FUNCTION_BLOCK SUBL_105_DRILLING-ROUND_HOLE (* 105-variable local group subscriber *)
  (* Standard: 61499-2 *)
  (* Version 1.0, 21-03-12, GASR, Universidade do Estado de Santa Catarina *)
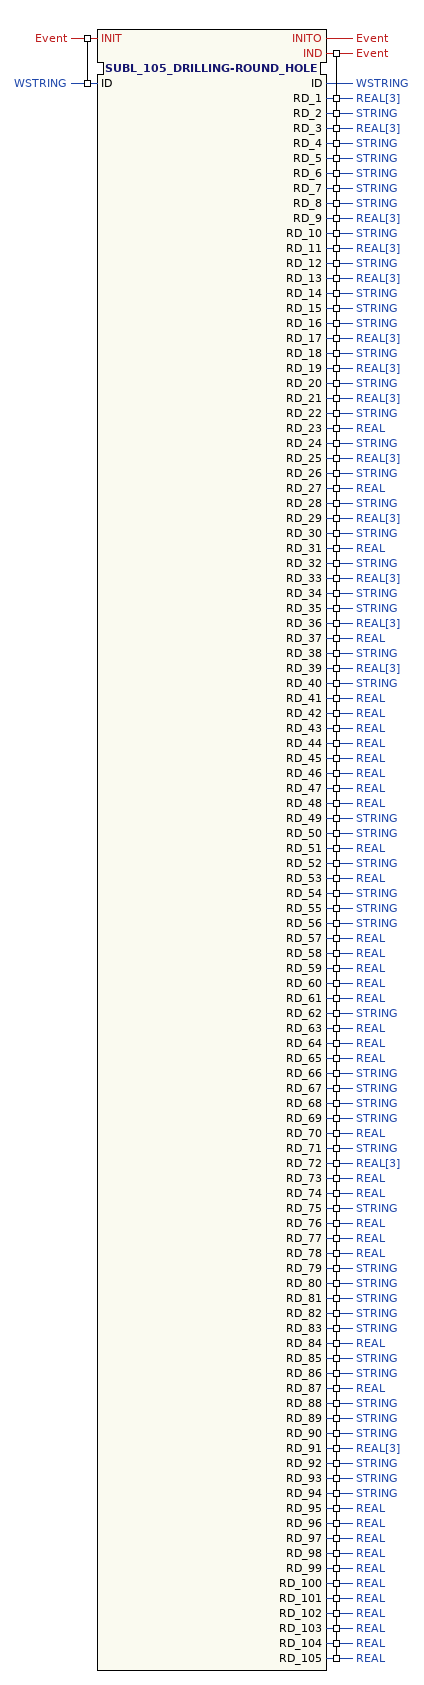
  EVENT_INPUT
    INIT WITH ID; (* Service Initialization *)
  END_EVENT
  EVENT_OUTPUT
    INITO; (* Initialization Confirm *)
    IND WITH RD_1, RD_2, RD_3, RD_4, RD_5, RD_6, RD_7, RD_8, RD_9, RD_10, RD_11, RD_12, RD_13, RD_14, RD_15, RD_16, RD_17, RD_18, RD_19, RD_20, RD_21, RD_22, RD_23, RD_24, RD_25, RD_26, RD_27, RD_28, RD_29, RD_30, RD_31, RD_32, RD_33, RD_34, RD_35, RD_36, RD_37, RD_38, RD_39, RD_40, RD_41, RD_42, RD_43, RD_44, RD_45, RD_46, RD_47, RD_48, RD_49, RD_50, RD_51, RD_52, RD_53, RD_54, RD_55, RD_56, RD_57, RD_58, RD_59, RD_60, RD_61, RD_62, RD_63, RD_64, RD_65, RD_66, RD_67, RD_68, RD_69, RD_70, RD_71, RD_72, RD_73, RD_74, RD_75, RD_76, RD_77, RD_78, RD_79, RD_80, RD_81, RD_82, RD_83, RD_84, RD_85, RD_86, RD_87, RD_88, RD_89, RD_90, RD_91, RD_92, RD_93, RD_94, RD_95, RD_96, RD_97, RD_98, RD_99, RD_100, RD_101, RD_102, RD_103, RD_104, RD_105; (* Service Indication *)
  END_EVENT
  VAR_INPUT
    ID : WSTRING; (* Default id is the FB instance name *)
  END_VAR
  VAR_OUTPUT
    ID : WSTRING; (* Default id is the FB instance name *)
    RD_1 : ARRAY [0..2] OF REAL; (* pos *)
    RD_2 : STRING; (* current_tool *)
    RD_3 : ARRAY [0..2] OF REAL; (* setup.Its_secplane.position.location.coordinates *)
    RD_4 : STRING; (* round_hole.its_id *)
    RD_5 : STRING; (* its_workpiece.its_id *)
    RD_6 : STRING; (* its_operations.its_id LIST - the list is concatenated in one string *)
    RD_7 : STRING; (* feature_placement.name *)
    RD_8 : STRING; (* feature_placement.location.name *)
    RD_9 : ARRAY [0..2] OF REAL; (* feature_placement.location.coordinates *)
    RD_10 : STRING; (* feature_placement.axis.its_id *)
    RD_11 : ARRAY [0..2] OF REAL; (* feature_placement.axis.direction_ratios *)
    RD_12 : STRING; (* feature_placement.ref_direction.its_id *)
    RD_13 : ARRAY [0..2] OF REAL; (* feature_placement.ref_direction_ratios *)
    RD_14 : STRING; (* depth.name *)
    RD_15 : STRING; (* depth.postion.name *)
    RD_16 : STRING; (* depth.position.location.name *)
    RD_17 : ARRAY [0..2] OF REAL; (* depth.position.location.coordinates *)
    RD_18 : STRING; (* depth.position.axis.its_id *)
    RD_19 : ARRAY [0..2] OF REAL; (* depth.position.axis.direction_ratios *)
    RD_20 : STRING; (* depth.position.ref_direction.its_id *)
    RD_21 : ARRAY [0..2] OF REAL; (* depth.position.ref_direction_ratios *)
    RD_22 : STRING; (* diameter *)
    RD_23 : REAL; (* diameter.theoretical_size *)
    RD_24 : STRING; (* diameter.implicit_tolerance *)
    RD_25 : ARRAY [0..2] OF REAL; (* diameter.{vector}, vector = {upper_limit, lower_limit, significant_digits} or {deviation,grade,its_fitting_type} *)
    RD_26 : STRING; (* change_in_diameter, "diameter_taper" or "angle_taper" *)
    RD_27 : REAL; (* change_in_diameter.theoretical_size *)
    RD_28 : STRING; (* change_in_diameter.implicit_tolerance *)
    RD_29 : ARRAY [0..2] OF REAL; (* change_in_diameter.{vector}, vector = {upper_limit, lower_limit, significant_digits} or {deviation,grade,its_fitting_type} *)
    RD_30 : STRING; (* bottom_condition, "through_bottom_condition" or ... *)
    RD_31 : REAL; (* bottom_condition.theoretical_size *)
    RD_32 : STRING; (* bottom_condition.implicit_tolerance *)
    RD_33 : ARRAY [0..2] OF REAL; (* bottom_condition.{vector}, vector = {upper_limit, lower_limit, significant_digits} or {deviation,grade,its_fitting_type} *)
    RD_34 : STRING; (* drilling.its_id *)
    RD_35 : STRING; (* its_toolpath.its_list *)
    RD_36 : ARRAY [0..2] OF REAL; (* its_tool_direction *)
    RD_37 : REAL; (* retract_plane *)
    RD_38 : STRING; (* start_point.name *)
    RD_39 : ARRAY [0..2] OF REAL; (* start_point.coordinates *)
    RD_40 : STRING; (* its_tool.its_id *)
    RD_41 : REAL; (* its_tool.its_tool_body.dimension.diameter *)
    RD_42 : REAL; (* its_tool.its_tool_body.dimension.tool_tip_half_angle *)
    RD_43 : REAL; (* its_tool.its_tool_body.dimension.tool_circumference_angle *)
    RD_44 : REAL; (* its_tool.its_tool_body.dimension.cutting_edge_lenght *)
    RD_45 : REAL; (* its_tool.its_tool_body.dimension.edge_radius *)
    RD_46 : REAL; (* its_tool.its_tool_body.dimension.edge_center_vertical *)
    RD_47 : REAL; (* its_tool.its_tool_body.dimension.edge_center_horizontal *)
    RD_48 : REAL; (* its_tool.its_tool_body.number_of_teeth *)
    RD_49 : STRING; (* its_tool.its_tool_body.hand_of_cut *)
    RD_50 : STRING; (* its_tool.its_tool_body.coolant_through *)
    RD_51 : REAL; (* its_tool.its_tool_body.pilot_length *)
    RD_52 : STRING; (* its_tool.its_tool_body.{other_tool_body_parameter} *)
    RD_53 : REAL; (* its_tool.its_cutting_edge.tool_offset_length *)
    RD_54 : STRING; (* its_tool.its_cutting_edge.its_material.standard_identifier *)
    RD_55 : STRING; (* its_tool.its_cutting_edge.its_material.material_identifier *)
    RD_56 : STRING; (* its_tool.its_cutting_edge.its_material.material_property.{list_of_parameters} *)
    RD_57 : REAL; (* its_tool.its_cutting_edge.its_technological_data.cutting_angle *)
    RD_58 : REAL; (* its_tool.its_cutting_edge.its_technological_data.free_angle *)
    RD_59 : REAL; (* its_tool.its_cutting_edge.its_technological_data.aux_angle *)
    RD_60 : REAL; (* its_tool.its_cutting_edge.expected_tool_life *)
    RD_61 : REAL; (* its_tool.its_cutting_edge.its_technology.feedrate *)
    RD_62 : STRING; (* its_tool.its_cutting_edge.its_technology.feedrate_reference *)
    RD_63 : REAL; (* its_tool.its_cutting_edge.its_technology.cutspeed *)
    RD_64 : REAL; (* its_tool.its_cutting_edge.its_technology.spindle *)
    RD_65 : REAL; (* its_tool.its_cutting_edge.its_technology.feedrate_per_tooth *)
    RD_66 : STRING; (* its_tool.its_cutting_edge.its_technology.sincronize_spindle_with_feed *)
    RD_67 : STRING; (* its_tool.its_cutting_edge.its_technology.inhibit_feedrate_override *)
    RD_68 : STRING; (* its_tool.its_cutting_edge.its_technology.inhibit_spindle_override *)
    RD_69 : STRING; (* its_tool.its_cutting_edge.its_technology.its_adaptive_control *)
    RD_70 : REAL; (* its_tool.overall_assembly_length *)
    RD_71 : STRING; (* its_tool.direction_for_spindle_orientation.its_id *)
    RD_72 : ARRAY [0..2] OF REAL; (* its_tool.direction_for_spindle_orientation.direction_ratios *)
    RD_73 : REAL; (* its_tool.tool_holder_diameter_for_spindle_orientation *)
    RD_74 : REAL; (* its_technology.feedrate *)
    RD_75 : STRING; (* its_technology.feedrate_reference *)
    RD_76 : REAL; (* its_technology.cutspeed *)
    RD_77 : REAL; (* its_technology.spindle *)
    RD_78 : REAL; (* its_technology.feedrate_per_tooth *)
    RD_79 : STRING; (* its_technology.sincronize_spindle_with_feed *)
    RD_80 : STRING; (* its_technology.inhibit_feedrate_override *)
    RD_81 : STRING; (* its_technology.inhibit_spindle_override *)
    RD_82 : STRING; (* its_technology.its_adaptive_control *)
    RD_83 : STRING; (* its_machine_functions.coolant *)
    RD_84 : REAL; (* its_machine_functions.coolant_pressure *)
    RD_85 : STRING; (* its_machine_functions.mist *)
    RD_86 : STRING; (* its_machine_functions.through_spindle_coolant *)
    RD_87 : REAL; (* its_machine_functions.through_pressure *)
    RD_88 : STRING; (* its_machine_functions.axis_clamping *)
    RD_89 : STRING; (* its_machine_functions.chip_removal *)
    RD_90 : STRING; (* its_machine_functions.oriented_spindle_stop.its_id *)
    RD_91 : ARRAY [0..2] OF REAL; (* its_machine_functions.oriented_spindle_stop.direction_ratios *)
    RD_92 : STRING; (* its_machine_functions.its_process_model.ini_data_file *)
    RD_93 : STRING; (* its_machine_functions.its_process_model.its_type *)
    RD_94 : STRING; (* its_machine_functions.other_functions *)
    RD_95 : REAL; (* overcut_length *)
    RD_96 : REAL; (* cutting_depth *)
    RD_97 : REAL; (* previous_diameter *)
    RD_98 : REAL; (* dwell_time_bottom *)
    RD_99 : REAL; (* feed_on_retract *)
    RD_100 : REAL; (* its_machining_strategy.reduced_cut_at_start *)
    RD_101 : REAL; (* its_machining_strategy.reduced_feed_at_start *)
    RD_102 : REAL; (* its_machining_strategy.depth_of_start *)
    RD_103 : REAL; (* its_machining_strategy.reduced_cut_at_end *)
    RD_104 : REAL; (* its_machining_strategy.reduced_feed_at_end *)
    RD_105 : REAL; (* its_machining_strategy.depth_of_end *)
  END_VAR
  SERVICE PUBL_105/SUBL_105 (* Data publication service *)
    SEQUENCE normal_establishment
      PUBL_105.INIT(ID) -> PUBL_105.INITO();
      SUBL_105.INIT(ID) -> SUBL_105.INITO();
    END_SEQUENCE
    SEQUENCE normal_data_transfer
      PUBL_105.REQ(SD_1,SD_2,SD_3,SD_4,SD_5,SD_6,SD_7,SD_8,SD_9,SD_10,SD_11,SD_12,SD_13,SD_14,SD_15,SD_16,SD_17,SD_18,SD_19,SD_20,SD_21,SD_22,SD_23,SD_24,SD_25,SD_26,SD_27,SD_28,SD_29,SD_30,SD_31,SD_32,SD_33,SD_34,SD_35,SD_36,SD_37,SD_38,SD_39,SD_40,SD_41,SD_42,SD_43,SD_44,SD_45,SD_46,SD_47,SD_48,SD_49,SD_50,SD_51,SD_52,SD_53,SD_54,SD_55,SD_56,SD_57,SD_58,SD_59,SD_60,SD_61,SD_62,SD_63,SD_64,SD_65,SD_66,SD_67,SD_68,SD_69,SD_70,SD_71,SD_72,SD_73,SD_74,SD_75,SD_76,SD_77,SD_78,SD_79,SD_80,SD_81,SD_82,SD_83,SD_84,SD_85,SD_86,SD_87,SD_88,SD_89,SD_90,SD_91,SD_92,SD_93,SD_94,SD_95,SD_96,SD_97,SD_98,SD_99,SD_100,SD_101,SD_102,SD_103,SD_104,SD_105) -> Subl_105.IND(RD_1,RD_2,RD_3,RD_4,RD_5,RD_6,RD_7,RD_8,RD_9,RD_10,RD_11,RD_12,RD_13,RD_14,RD_15,RD_16,RD_17,RD_18,RD_19,RD_20,RD_21,RD_22,RD_23,RD_24,RD_25,RD_26,RD_27,RD_28,RD_29,RD_30,RD_31,RD_32,RD_33,RD_34,RD_35,RD_36,RD_37,RD_38,RD_39,RD_40,RD_41,RD_42,RD_43,RD_44,RD_45,RD_46,RD_47,RD_48,RD_49,RD_50,RD_51,RD_52,RD_53,RD_54,RD_55,RD_56,RD_57,RD_58,RD_59,RD_60,RD_61,RD_62,RD_63,RD_64,RD_65,RD_66,RD_67,RD_68,RD_69,RD_70,RD_71,RD_72,RD_73,RD_74,RD_75,RD_76,RD_77,RD_78,RD_79,RD_80,RD_81,RD_82,RD_83,RD_84,RD_85,RD_86,RD_87,RD_88,RD_89,RD_90,RD_91,RD_92,RD_93,RD_94,RD_95,RD_96,RD_97,RD_98,RD_99,RD_100,RD_101,RD_102,RD_103,RD_104,RD_105);
    END_SEQUENCE
  END_SERVICE
END_FUNCTION_BLOCK
